{attribute 'enable_dynamic_creation'}
FUNCTION_BLOCK FB_XmlLogger IMPLEMENTS ILogger
VAR_INPUT
END_VAR
VAR_OUTPUT
END_VAR
VAR
END_VAR

METHOD PUBLIC Write : STRING
VAR_INPUT
	sMsg      : STRING;
END_VAR
Write := CONCAT('xml-', sMsg);
// open xml file
// write the message into the xml file
// close xml file
END_METHOD

END_FUNCTION_BLOCK

(* stored: Version 1.1.0.1, ProductVersion 3.1.0.24
   POU FB_XmlLogger: Id {142f02b9-70fe-4235-8d7b-5808e6dd12dc}
   Method Write: Id {88070c92-1819-408a-9ef0-7aa749e9dc72} *)
